Omron CX-Programmer project NewProject (CX-Programmer 9.73)

# PLC NewPLC1: CP1E N20

## Global symbols (name address type ; comment)
0.01 BOOL  ; pb start
0.02 BOOL  ; sensor 1
0.03 BOOL  ; sensor 2
0.06 BOOL  ; pb stop
100.01 BOOL  ; solenoid a
100.02 BOOL  ; motor 1
100.05 BOOL  ; solenoid b
200.00 BOOL  ; relay
C001 BOOL  ; counter
T001 BOOL  ; timer1

## Program NewProgram1 (cyclic task 0)

### Section Section1

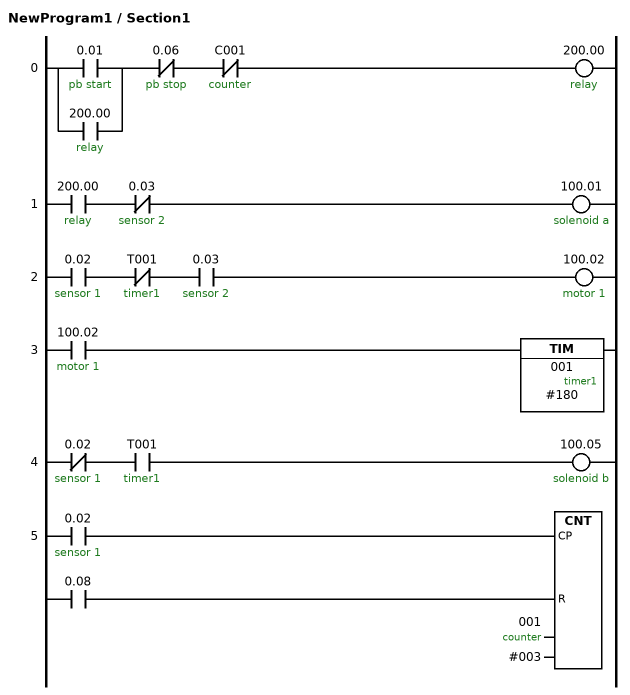
; rung 0
LD 0.01  ; pb start
OR 200.00  ; relay
ANDNOT 0.06  ; pb stop
ANDNOT C001  ; counter
OUT 200.00  ; relay
; rung 1
LD 200.00  ; relay
ANDNOT 0.03  ; sensor 2
OUT 100.01  ; solenoid a
; rung 2
LD 0.02  ; sensor 1
ANDNOT T001  ; timer1
AND 0.03  ; sensor 2
OUT 100.02  ; motor 1
; rung 3
LD 100.02  ; motor 1
TIM 001 #180  ; timer1
; rung 4
LDNOT 0.02  ; sensor 1
AND T001  ; timer1
OUT 100.05  ; solenoid b
; rung 5
LD 0.02  ; sensor 1
LD 0.08
CNT 001 #003  ; counter

### Section END
; rung 0
END(001)